Universal Robots PolyScope program: andrea8.urp

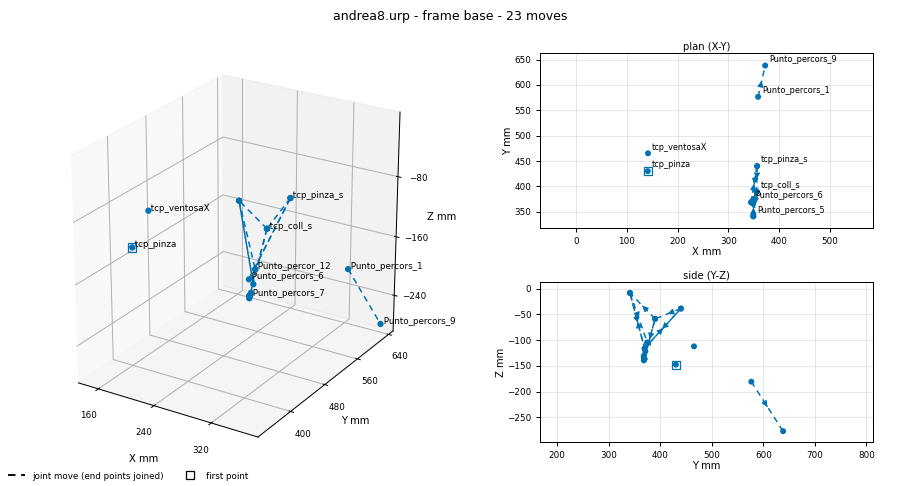
[picture p0: tool path of andrea8.urp in frame base, 23 of 31 moves have a stored position in this frame; points joined in program order, loops and branches not executed]
Program andrea8 (installation=Kong_install82 directory=/programs/usbdisk/andrea8 createdIn=3.15.4.106291 lastSavedIn=3.15.4.106291 robotSerialNumber=2017357596)
Calibrated DH parameters: a=[0.000104, -0.381245, -0.385946, 0.00002, 0.000083, 0]; d=[0.089177, 59.99214, -36.297918, -23.584132, 0.094784, 0.082552]; alpha=[1.570197, -0.003145, 0.002952, 1.570494, -1.570091, 0]; deltaTheta=[-0.00001, -0.459739, 0.638868, -0.17972, -0.000006, -0.000462]
InitVariablesNode variables(variable(name=XY, expression=[0,0]), variable(name=ant, expression=3), variable(name=col, expression=4), variable(name=ghr, expression=2), variable(name=nCycle, expression=0), variable(name=nfc, expression=1), variable(name=pallStocks, expression=[16,16,16,40,16,16,16,40,16,16,16,40,16,40,0,0]), variable(name=pick, expression=[0,0]))
Robot Program (runOnlyOnce=false)
  Script file /programs/usbdisk/andrea8/nuova dir/relPose.script
    | def relPose(FeaturePose,vect):
    | 
    |     # FeaturePose is the pose for the feature
    |     # vect = p[0.1, 0, 0, 0, 0, 0] makes us move 10cm in the X direction of the feature
    |     # credits: https://forum.universal-robots.com/t/move-tcp-relative-to-feature/15492
    | 
    |    PoseRelativeToFeature = pose_trans(pose_inv(FeaturePose), get_actual_tcp_pose())
    |    MoveTCPRelativeToFeature = pose_add(PoseRelativeToFeature, vect)
    |    return pose_trans(FeaturePose, MoveTCPRelativeToFeature)
    | 
    | end
  Script file /programs/usbdisk/andrea8/tcpMov.script
    | def tcpMov(vect):
    | 
    |     # FeaturePose is the pose for the feature
    |     # vect = p[0.1, 0, 0, 0, 0, 0] makes us move 10cm in the X direction of the feature
    |     # credits: https://forum.universal-robots.com/t/move-tcp-relative-to-feature/15492
    | 
    |    tcp_pose = get_actual_tcp_pose()
    |    return pose_add(tcp_pose, vect)
    | 
    | 
    | end
  Script file /programs/usbdisk/andrea8/calcItemPosition.script
    | def calcItemPosition(pick, item, pallDefs, grid, featOrigin):
    | 
    |     # calcola la posizione assoluta del pezzo scelto da pickPalletItem
    | 
    |     # nPosX è il numero di colonne
    |     # nPosY è il numero di righe
    |     # distX è la distanza tra colonne
    |     # distY è la distanza tra righe
    |     # [posX1, posY1] è la posizione del primo pezzo rispetto all'origine del pallet
    | 
    |     nPallet = pick[0] + 1 # numero del pallet (gli id partono da 0)
    |     nItem = pick[1] + 1 # numero del pezzo
    | 
    |     nPosXgrid = grid[0] # numero di posizioni della giglia in X
    |     distXgrid = grid[2] # distanza tra gli slot della griglia in X
    |     distYgrid = grid[3] # distanza tra gli slot della griglia in Y
    | 
    |     pallPosX = nPallet%nPosXgrid
    |     if(pallPosX==0): pallPosX = nPosXgrid end
    |     pallPosY = ceil(nPallet/nPosXgrid)
    | 
    |     pallPosX1 = grid[4]
    |     pallPosY1 = grid[5]
    | 
    | 
    |     nPosX = pallDefs[item,0]
    |     nPosY = pallDefs[item,1]
    |     distX = pallDefs[item,2]
    |     distY = pallDefs[item,3]
    |     posX1 = pallDefs[item,4]
    |     posY1 = pallDefs[item,5]
    | 
    |     posX = nItem%nPosX
    |     if(posX==0): posX = nPosX end
    |     posY = ceil(nItem/nPosX)
    | 
    |     # [X,Y] è la posizione del pezzo rispetto all'origine della griglia
    | 
    |     X=distX*(posX - 1) + posX1 + distXgrid*(pallPosX - 1) + pallPosX1
    |     Y=distY*(posY - 1) + posY1 + distYgrid*(pallPosY - 1) + pallPosY1
    |     xy=[X,Y]
    | 
    |     return xy
    | 
    |  end
  Script file /programs/usbdisk/andrea8/pickPalletItem.script
    | def pickPalletItem(type, pallDefs, pallTypes, pallStocks):
    | 
    |   # seleziona un pezzo sulla griglia, noti il tipo di pezzo e lo stato della griglia
    | 
    |   # lo script funziona finché le variabili del robot non vengono resettate. Tuttavia, anche
    |   # in caso di riavvio, è possibile scrivere manualmente le info sulla griglia e lo stock
    |   # all'inizio del programma, così da 'insegnare' al robot dove farlo
    |   # riprendere
    | 
    |   iPallet = 0 # inizializzo l'id del pallet
    | 
    |   while iPallet < length(pallStocks):
    | 
    |     if pallTypes[iPallet] == type and pallStocks[iPallet] > 0 :
    | 
    |       nItems = pallStocks[iPallet] # numero di pezzi nello stock del pallet iesimo
    | 
    |       nPosX = pallDefs[type,0] # numero di posizioni lungo x, come definito per il pallet di tipo "type"
    |       nPosY = pallDefs[type,1] # numero di posizioni lungo y, come definito per il pallet di tipo "type"
    | 
    |       stockMax = nPosX*nPosY
    |       iItem = stockMax - nItems # id del pezzo
    | 
    |       pick = [iPallet,iItem]
    | 
    |       # pick = [id del pallet, id del pezzo]
    | 
    |       return pick
    |  end
    | iPallet = iPallet + 1
    | end
    | end
  Script file /programs/usbdisk/andrea8/stockUpdate.script
    | def stockUpdate(pick,stock):
    | 
    |     # simple function that ingests the output of pickItem and returns the
    |     # modified stock array. just so to avoid using global variables and
    |     # multi-dimensional arrays
    | 
    |     i = pick[0]
    |     stock[i] = stock[i] - 1
    |     return stock
    | 
    | 
    | end
  SuppressedNode
    Script file /programs/usbdisk/andrea8/ini_grids.script
      | def ini_grids():
      | 
      |     # grid = [nPallPosX, nPallPosY, distPallX, distPallY, pallPosX1, pallPosY1, pallPosZ1]
      |     # la struttura e' del tutto analoga in logica con quella espressa in defs
      |     grids = [
      |                      [4, 4, 90, 90, 10, 20, 6] # griglia moduli
      |                      [2, 1, 200, 0, 20, -40, 45] # griglia stazioni
      |                  ]
      |     return grids
      | end
  Script file /programs/usbdisk/andrea8/ini_grid.script
    | def ini_grid():
    | 
    |     # grid = [nPallPosX, nPallPosY, distPallX, distPallY, pallPosX1, pallPosY1, pallPosZ1]
    |     # la struttura e' del tutto analoga in logica con quella espressa in defs
    |     grid = [4, 4, 90, 90, 10, 17.5, 6]
    |     return grid
    | end
  Script file /programs/usbdisk/andrea8/ini_defs.script
    | def ini_defs():
    | 
    |     # definition = [nPosX,nPosY,distX,distY,posX1,posY1,posZ1]
    | 
    |     # nPosX è il numero di colonne
    |     # nPosY è il numero di righe
    |     # distX è la distanza tra colonne
    |     # distY è la distanza tra righe
    |     # [posX1, posY1] è la posizione del primo pezzo rispetto all'origine del pallet
    |     # posZ1 e' la posizione che deve raggiungere il TCP lungo asse Z, che sarebbe asse verticale
    | 
    |     defs = [
    |         [0, 0, 0, 0, 0, 0, 0], # slot vuoto
    |         [4, 10, 18, 8, 11.5, 3.5, 11.1], # pallet nfc
    |         [4, 4, 21, 21, 5.5, 8.5, 49], # pallet ghiere
    |         [1, 1, 0, 0, 132.06, 44, 16.05], # stazione antenna
    |         [1, 2, 0, 40, 20.256, 24, 27.85] # stazione incollaggio
    |     ]
    |     return defs
    | end
  Script file /programs/usbdisk/andrea8/ini_types.script
    | def ini_types():
    | 
    |     visualTypes = [
    | 
    |         [0,0,0,0],
    |         [0,ghr,0,0],
    |         [0,0,0,nfc],
    |         [0,ghr,0,0]
    | 
    |     ]
    | 
    | # purtroppo fare questa array vuota di dimensione (righe)x(colonne) per aggirare le limitazioni di UR
    | # bisogna ricordarsi di cambiare questa dichiarazione di types se si cambia dimensione griglia
    | 
    |      types = [0,0,0,0,0,0,0,0,0,0,0,0,0,0,0,0]
    | 
    |     iii = 0
    |     s = size(visualTypes)
    |     i = 0
    |     while i < s[0]:
    | 
    |         ii=0
    |         while ii < s[1]:
    | 
    |             types[iii] = visualTypes[s[0]-1-i,ii]
    |             ii = ii + 1
    |             iii = iii + 1
    |         end
    |     i = i + 1
    |     end
    |     return types
    | end
  Script file /programs/usbdisk/andrea8/ini_stocks2.script
    | def ini_stocks(defs, types):
    | 
    |     global f = -1 # usa questo carattere per inizializzare automaticamente pallet pieni
    | 
    |     visualStocks = [
    | 
    |         [f, f, f, f],
    |         [f, f, f, f],
    |         [f, f, f, 36],
    |         [f ,f, f, f]
    | 
    |     ]
    | 
    | # purtroppo fare questa array vuota di dimensione (righe)x(colonne) per aggirare le limitazioni di UR
    | # bisogna ricordarsi di cambiare questa dichiarazione di types se si cambia dimensione griglia
    | 
    |      stocks = [0,0,0,0,0,0,0,0,0,0,0,0,0,0,0,0]
    | 
    |     iii = 0
    |     s = size(visualStocks)
    |     i = 0
    |     while i < s[0]:
    | 
    |         ii=0
    |         while ii < s[1]:
    |             if visualStocks[s[0]-1-i,ii] == f:
    |                 nPosX = defs[types[iii], 0]
    |                 nPosY = defs[types[iii], 1]
    |                 stocks[iii] = nPosX*nPosY
    |             else:
    | 
    |                 stocks[iii] = visualStocks[s[0]-1-i,ii]
    |             end
    |             ii = ii + 1
    |             iii = iii + 1
    |         end
    |     i = i + 1
    |     end
    |     return stocks
    | end
  If nCycle≟0
    Set NoAction
    pallTypes := ini_types()
    grid := ini_grid()
    pallDefs := ini_defs()
    pallStocks := ini_stocks(pallDefs,pallTypes)
    SuppressedNode
      Popup Message (haltProgram=false inputType=Variable) variable=grid
    ghr := ghr
    nfc := nfc
    ant := ant
    col := col
    URCap Open Gripper (SCHUNK End-of-Arm Modular System for UR, SCHUNK GmbH & Co.)
    nCycle := 1
    Wait Sleep waitTime=5
  MoveJ speed 60 deg/s, acceleration 80 deg/s^2 (useActiveTCP=false) tcp=Pinza
    Waypoint tcp_pinza: TCP in base x=141.498 y=430.173 z=-147.715 mm, rx=-2.3787 ry=0.7214 rz=1.7108 rad; joints [-125.948, -50.519, 103.828, -113.29, -23.958, -21.608] deg; pose in feature x=-0.012 y=-0.048 z=150.016 mm, rx=-1.1212 ry=1.1212 rz=0.4102 rad; flange x=182.463 y=570.54 z=26.56 mm, rx=-2.3787 ry=0.7214 rz=1.7108 rad
    item := ghr
    pick := pickPalletItem(item,pallDefs,pallTypes,pallStocks)
    SuppressedNode
      Popup Message (haltProgram=false inputType=Variable) variable=pick
    XY := calcItemPosition(pick, item,pallDefs, grid,piano_moduli)
    p_pall := relPose(piano_moduli,p[XY[0]/1000,XY[1]/1000,0.0,0.0,0.0,0.0])
    SuppressedNode
      Popup Message (haltProgram=false inputType=Variable) variable=XY
    Waypoint Punto_percors (Variable): variable=p_pall
  MoveJ speed 60 deg/s, acceleration 80 deg/s^2 (useActiveTCP=false) tcp=Pinza
    p_pezzo := relPose(piano_moduli,p[0.0, 0.0, -130*0.001, 0.0, 0.0, 0.0])
    Waypoint Punto_percors (Variable): variable=p_pezzo
    URCap Close Gripper (SCHUNK End-of-Arm Modular System for UR, SCHUNK GmbH & Co.)
    p_pezzo := relPose(piano_moduli,p[0.0, 0.0, 130/1000, 0.0, 0.0, 0.0])
    Waypoint Punto_percors (Variable): variable=p_pezzo
    pallStocks := stockUpdate(pick,pallStocks)
    SuppressedNode
      Popup Message (haltProgram=false inputType=Variable) variable=pallStocks
  MoveJ speed 60 deg/s, acceleration 80 deg/s^2 (useActiveTCP=false) tcp=Ventosa
    Waypoint tcp_ventosaX: TCP in base x=141.953 y=465.356 z=-112.213 mm, rx=-2.2886 ry=-0.6046 rz=-0.263 rad; joints [-121.609, -49.485, 100.63, -2.12, 68.781, 127.146] deg; flange x=141.931 y=500.256 z=-13.059 mm, rx=-2.2886 ry=-0.6046 rz=-0.263 rad
    SuppressedNode
      Waypoint tcp_ventosaY_s: TCP in base x=355.984 y=389.916 z=-58.857 mm, rx=-1.401 ry=-1.0647 rz=1.3858 rad; joints [-146.472, -36.177, 73.345, -37.097, -55.375, 194.745] deg; pose in feature x=141.985 y=465.345 z=-112.215 mm, rx=-1.4011 ry=-1.0646 rz=1.3857 rad; flange x=401.93 y=456.119 z=8.64 mm, rx=-1.401 ry=-1.0647 rz=1.3858 rad
    item := nfc
    pick := pickPalletItem(item,pallDefs,pallTypes,pallStocks)
    SuppressedNode
      Popup Message (haltProgram=false inputType=Variable) variable=pick
    XY := calcItemPosition(pick, item,pallDefs, grid,piano_moduli)
    p_pall := relPose(piano_moduli,p[XY[0]/1000,XY[1]/1000,0.0,0.0,0.0,0.0])
    SuppressedNode
      Popup Message (haltProgram=false inputType=Variable) variable=XY
    Waypoint Punto_percors (Variable): variable=p_pall
  MoveJ speed 60 deg/s, acceleration 80 deg/s^2 (useActiveTCP=false) tcp=Ventosa
    p_pezzo := relPose(piano_moduli,p[0.0, 0.0, -181.4*0.001, 0.0, 0.0, 0.0])
    Waypoint Punto_percors (Variable): variable=p_pezzo
    Wait Sleep waitTime=2
    p_pezzo := relPose(piano_moduli,p[0.0, 0.0, 181.4/1000, 0.0, 0.0, 0.0])
    Waypoint Punto_percors (Variable): variable=p_pezzo
    pallStocks := stockUpdate(pick,pallStocks)
    SuppressedNode
      Popup Message (haltProgram=false inputType=Variable) variable=pallStocks
  MoveJ speed 60 deg/s, acceleration 80 deg/s^2 (useActiveTCP=false) tcp=Ventosa
    Waypoint Punto_percors_1: TCP in base x=358.691 y=576.543 z=-180.701 mm, rx=-2.2887 ry=-0.6045 rz=-0.2628 rad; joints [-132.678, -21.575, 54.335, 20.288, 61.783, 117.598] deg; flange x=358.684 y=611.454 z=-81.55 mm, rx=-2.2887 ry=-0.6045 rz=-0.2628 rad
    Waypoint Punto_percors_9: TCP in base x=372.703 y=638.173 z=-276.765 mm, rx=-2.2781 ry=-0.6995 rz=-0.1741 rad; joints [-130.314, 4.573, 13.616, 38.475, 59.716, 114.972] deg; flange x=372.486 y=675.646 z=-178.554 mm, rx=-2.2781 ry=-0.6995 rz=-0.1741 rad
    SuppressedNode
      MoveJ speed 60 deg/s, acceleration 80 deg/s^2 (useActiveTCP=true)
        Waypoint Punto_percors_2: 
  MoveJ speed 60 deg/s, acceleration 80 deg/s^2 (useActiveTCP=false) tcp=Ventosa
    p_pezzo := relPose(piano_moduli,p[0.0, 0.0, -55*0.001, 0.0, 0.0, 0.0])
    Waypoint Punto_percors (Variable): variable=p_pezzo
    Wait Sleep waitTime=2
    p_pezzo := relPose(piano_moduli,p[0.0, 0.0, 55/1000, 0.0, 0.0, 0.0])
    Waypoint Punto_percors (Variable): variable=p_pezzo
  MoveJ speed 60 deg/s, acceleration 80 deg/s^2 (useActiveTCP=false) tcp=Pinza
    Waypoint tcp_pinza_s: TCP in base x=356.783 y=439.979 z=-38.857 mm, rx=1.9379 ry=-1.1643 rz=-1.0823 rad; joints [-132.207, -20.407, 45.734, -60.67, -53.979, 1] deg; flange x=387.119 y=665.322 z=-46.123 mm, rx=1.9379 ry=-1.1643 rz=-1.0823 rad
    Waypoint Punto_percors_6: TCP in base x=344.955 y=369.152 z=-116.441 mm, rx=1.9235 ry=-1.2186 rz=-1.1045 rad; joints [-136.086, -22.163, 63.024, -76.094, -54.959, 0.389] deg; flange x=386.118 y=592.787 z=-123.208 mm, rx=1.9235 ry=-1.2186 rz=-1.1045 rad
    URCap Open Gripper (SCHUNK End-of-Arm Modular System for UR, SCHUNK GmbH & Co.)
    Waypoint tcp_pinza_s: TCP in base x=356.783 y=439.979 z=-38.857 mm, rx=1.9379 ry=-1.1643 rz=-1.0823 rad; joints [-132.207, -20.407, 45.734, -60.67, -53.979, 1] deg; flange x=387.119 y=665.322 z=-46.123 mm, rx=1.9379 ry=-1.1643 rz=-1.0823 rad
  SuppressedNode
    MoveJ speed 60 deg/s, acceleration 80 deg/s^2 (useActiveTCP=false) tcp=Pinza
      p_pezzo := relPose(piano_moduli,p[0.0, 0.0, -100*0.001, 0.0, 0.0, 0.0])
      Waypoint Punto_percors (Variable): variable=p_pezzo
      p_pezzo := relPose(piano_moduli,p[0.0, 0.0, 100/1000, 0.0, 0.0, 0.0])
      Waypoint Punto_percors (Variable): variable=p_pezzo
  MoveJ speed 60 deg/s, acceleration 80 deg/s^2 (useActiveTCP=false) tcp=Dosatore_Colla
    Waypoint tcp_coll_s: TCP in base x=355.98 y=389.944 z=-58.821 mm, rx=-0.0221 ry=-3.1138 rz=0.4025 rad; joints [-139.161, -64.308, 106.34, -121.985, -100.827, 102.96] deg; flange x=356.624 y=435.245 z=113.503 mm, rx=0.7684 ry=-2.9515 rz=0.3801 rad
    Waypoint Punto_percors_7: TCP in base x=346.196 y=368.904 z=-136.542 mm, rx=-0.022 ry=-3.1138 rz=0.4025 rad; joints [-139.88, -59.505, 111.836, -132.417, -100.987, 102.258] deg; flange x=346.894 y=417.717 z=49.148 mm, rx=0.7685 ry=-2.9514 rz=0.38 rad
    Waypoint Punto_percors_8: TCP in base x=346.193 y=368.067 z=-139.507 mm, rx=-0.0222 ry=-3.1137 rz=0.4027 rad; joints [-139.945, -59.217, 112.004, -132.878, -101.004, 102.201] deg; flange x=346.901 y=416.902 z=46.177 mm, rx=0.7683 ry=-2.9514 rz=0.3802 rad
    Waypoint Punto_percors_7: TCP in base x=346.196 y=368.904 z=-136.542 mm, rx=-0.022 ry=-3.1138 rz=0.4025 rad; joints [-139.88, -59.505, 111.836, -132.417, -100.987, 102.258] deg; flange x=346.894 y=417.717 z=49.148 mm, rx=0.7685 ry=-2.9514 rz=0.38 rad
    Waypoint arco01: TCP in base x=346.236 y=368.89 z=-136.518 mm, rx=-0.0959 ry=-3.05 rz=0.3936 rad; joints [-141.187, -58.835, 109.658, -128.209, -98.558, 103.729] deg; flange x=360.097 y=417.145 z=48.801 mm, rx=0.6834 ry=-2.9135 rz=0.3475 rad
    Waypoint arco02: motionParameters(blendRadius=0); TCP in base x=346.216 y=368.872 z=-136.545 mm, rx=-0.179 ry=-2.9723 rz=0.3829 rad; joints [-142.748, -57.872, 107.148, -123.504, -95.68, 105.297] deg; flange x=375.525 y=415.536 z=47.377 mm, rx=0.5857 ry=-2.8653 rz=0.31 rad
    Waypoint arco03: motionParameters(blendRadius=0); TCP in base x=346.203 y=368.894 z=-136.515 mm, rx=-0.2657 ry=-2.8849 rz=0.3708 rad; joints [-144.474, -56.651, 104.495, -118.647, -92.526, 106.837] deg; flange x=392.12 y=412.637 z=44.709 mm, rx=0.482 ry=-2.8087 rz=0.2699 rad
    SuppressedNode
      Waypoint arco04: motionParameters(blendRadius=0); TCP in base x=346.203 y=368.881 z=-136.572 mm, rx=-0.3164 ry=-2.8302 rz=0.3633 rad; joints [-145.538, -55.821, 102.932, -115.817, -90.6, 107.69] deg; flange x=402.069 y=410.254 z=42.401 mm, rx=0.4203 ry=-2.7721 rz=0.2459 rad
    SuppressedNode
      Waypoint arrco05: motionParameters(blendRadius=0); TCP in base x=346.234 y=368.906 z=-136.515 mm, rx=-0.3852 ry=-2.7521 rz=0.3526 rad; joints [-147.033, -54.592, 100.815, -111.993, -87.907, 108.809] deg; flange x=415.666 y=406.217 z=38.559 mm, rx=0.3354 ry=-2.7188 rz=0.2129 rad
    SuppressedNode
      Waypoint arco06: motionParameters(blendRadius=0); TCP in base x=346.215 y=368.872 z=-136.573 mm, rx=-0.447 ry=-2.677 rz=0.3424 rad; joints [-148.443, -53.359, 98.932, -108.559, -85.383, 109.759] deg; flange x=427.962 y=401.606 z=34.043 mm, rx=0.2577 ry=-2.666 rz=0.1826 rad
    SuppressedNode
      Waypoint arco07: motionParameters(blendRadius=0); TCP in base x=346.221 y=368.89 z=-136.541 mm, rx=-0.508 ry=-2.5984 rz=0.3316 rad; joints [-149.891, -52.049, 97.106, -105.173, -82.796, 110.659] deg; flange x=440.036 y=396.148 z=28.747 mm, rx=0.1797 ry=-2.6097 rz=0.1519 rad
    SuppressedNode
      Waypoint arco08: motionParameters(blendRadius=0); TCP in base x=346.175 y=368.881 z=-136.554 mm, rx=-0.5601 ry=-2.5271 rz=0.322 rad; joints [-151.177, -50.841, 95.583, -102.267, -80.5, 111.395] deg; flange x=450.208 y=390.667 z=23.341 mm, rx=0.1118 ry=-2.5574 rz=0.1253 rad
    SuppressedNode
      Waypoint arco07: motionParameters(blendRadius=0); TCP in base x=346.221 y=368.89 z=-136.541 mm, rx=-0.508 ry=-2.5984 rz=0.3316 rad; joints [-149.891, -52.049, 97.106, -105.173, -82.796, 110.659] deg; flange x=440.036 y=396.148 z=28.747 mm, rx=0.1797 ry=-2.6097 rz=0.1519 rad
    SuppressedNode
      Waypoint arco06: motionParameters(blendRadius=0); TCP in base x=346.215 y=368.872 z=-136.573 mm, rx=-0.447 ry=-2.677 rz=0.3424 rad; joints [-148.443, -53.359, 98.932, -108.559, -85.383, 109.759] deg; flange x=427.962 y=401.606 z=34.043 mm, rx=0.2577 ry=-2.666 rz=0.1826 rad
    SuppressedNode
      Waypoint arrco05: motionParameters(blendRadius=0); TCP in base x=346.234 y=368.906 z=-136.515 mm, rx=-0.3852 ry=-2.7521 rz=0.3526 rad; joints [-147.033, -54.592, 100.815, -111.993, -87.907, 108.809] deg; flange x=415.666 y=406.217 z=38.559 mm, rx=0.3354 ry=-2.7188 rz=0.2129 rad
    SuppressedNode
      Waypoint arco04: motionParameters(blendRadius=0); TCP in base x=346.203 y=368.881 z=-136.572 mm, rx=-0.3164 ry=-2.8302 rz=0.3633 rad; joints [-145.538, -55.821, 102.932, -115.817, -90.6, 107.69] deg; flange x=402.069 y=410.254 z=42.401 mm, rx=0.4203 ry=-2.7721 rz=0.2459 rad
    SuppressedNode
      Waypoint arco03: motionParameters(blendRadius=0); TCP in base x=346.203 y=368.894 z=-136.515 mm, rx=-0.2657 ry=-2.8849 rz=0.3708 rad; joints [-144.474, -56.651, 104.495, -118.647, -92.526, 106.837] deg; flange x=392.12 y=412.637 z=44.709 mm, rx=0.482 ry=-2.8087 rz=0.2699 rad
    Waypoint arco02: motionParameters(blendRadius=0); TCP in base x=346.216 y=368.872 z=-136.545 mm, rx=-0.179 ry=-2.9723 rz=0.3829 rad; joints [-142.748, -57.872, 107.148, -123.504, -95.68, 105.297] deg; flange x=375.525 y=415.536 z=47.377 mm, rx=0.5857 ry=-2.8653 rz=0.31 rad
    Waypoint arco01: TCP in base x=346.236 y=368.89 z=-136.518 mm, rx=-0.0959 ry=-3.05 rz=0.3936 rad; joints [-141.187, -58.835, 109.658, -128.209, -98.558, 103.729] deg; flange x=360.097 y=417.145 z=48.801 mm, rx=0.6834 ry=-2.9135 rz=0.3475 rad
    Waypoint tcp_coll_s: TCP in base x=355.98 y=389.944 z=-58.821 mm, rx=-0.0221 ry=-3.1138 rz=0.4025 rad; joints [-139.161, -64.308, 106.34, -121.985, -100.827, 102.96] deg; flange x=356.624 y=435.245 z=113.503 mm, rx=0.7684 ry=-2.9515 rz=0.3801 rad
    SuppressedNode
      Waypoint tcp_colla: TCP in base x=141.953 y=465.356 z=-112.213 mm, rx=-0.0207 ry=-2.9002 rz=1.1933 rad; joints [-112.251, -46.475, 88.048, -88.757, -104.681, 134.691] deg; flange x=143.75 y=590.738 z=14.373 mm, rx=0.6882 ry=-2.6438 rz=1.0836 rad
  MoveJ speed 60 deg/s, acceleration 80 deg/s^2 (useActiveTCP=false) tcp=Ventosa
    Waypoint Punto_percors_5: TCP in base x=349.319 y=341.12 z=-8.564 mm, rx=-1.0185 ry=-1.3146 rz=1.0001 rad; joints [-153.414, -49.535, 86.3, -36.662, -62.309, 164.702] deg; flange x=394.672 y=364.631 z=83.305 mm, rx=-1.0185 ry=-1.3146 rz=1.0001 rad
    Waypoint Punto_percor_11: TCP in base x=349.675 y=371.112 z=-122.13 mm, rx=-1.0185 ry=-1.3145 rz=1.0002 rad; joints [-150.91, -37.388, 83.592, -46.127, -59.801, 164.771] deg; flange x=395.037 y=394.636 z=-30.269 mm, rx=-1.0185 ry=-1.3145 rz=1.0002 rad
    Wait Sleep waitTime=1
    Waypoint Punto_percors_5: TCP in base x=349.319 y=341.12 z=-8.564 mm, rx=-1.0185 ry=-1.3146 rz=1.0001 rad; joints [-153.414, -49.535, 86.3, -36.662, -62.309, 164.702] deg; flange x=394.672 y=364.631 z=83.305 mm, rx=-1.0185 ry=-1.3146 rz=1.0001 rad
    SuppressedNode
      Waypoint tcp_ventosaY_s: TCP in base x=355.984 y=389.916 z=-58.857 mm, rx=-1.401 ry=-1.0647 rz=1.3858 rad; joints [-146.472, -36.177, 73.345, -37.097, -55.375, 194.745] deg; flange x=401.93 y=456.119 z=8.64 mm, rx=-1.401 ry=-1.0647 rz=1.3858 rad
    SuppressedNode
      Waypoint Punto_percors_4: 
  MoveJ speed 60 deg/s, acceleration 80 deg/s^2 (useActiveTCP=false) tcp=Pressa
    Waypoint Punto_percor_12: TCP in base x=349.834 y=374.867 z=-104.947 mm, rx=0.1982 ry=-1.5625 rz=-0.2204 rad; joints [-149.184, -43.549, 79.977, -36.342, -58.078, 74.726] deg; flange x=395.431 y=416.173 z=54.625 mm, rx=0.1982 ry=-1.5625 rz=-0.2204 rad
    Waypoint Punto_percor_13: TCP in base x=348.512 y=367.85 z=-131.982 mm, rx=0.1982 ry=-1.5627 rz=-0.2205 rad; joints [-149.684, -41.891, 81.658, -39.702, -58.567, 74.74] deg; flange x=394.082 y=409.131 z=27.605 mm, rx=0.1982 ry=-1.5627 rz=-0.2205 rad
    Wait Sleep waitTime=2
    Waypoint Punto_percor_12: TCP in base x=349.834 y=374.867 z=-104.947 mm, rx=0.1982 ry=-1.5625 rz=-0.2204 rad; joints [-149.184, -43.549, 79.977, -36.342, -58.078, 74.726] deg; flange x=395.431 y=416.173 z=54.625 mm, rx=0.1982 ry=-1.5625 rz=-0.2204 rad
    SuppressedNode
      Waypoint tcp_pressaY: TCP in base x=141.469 y=430.16 z=-147.709 mm, rx=-0.2128 ry=-1.5595 rz=0.1907 rad; joints [-127.014, -38.383, 85.876, -47.443, -35.896, 104.766] deg; flange x=188.109 y=545.63 z=-30.49 mm, rx=-0.2128 ry=-1.5595 rz=0.1907 rad
    SuppressedNode
      Waypoint tcp_pressaX: TCP in base x=141.415 y=430.194 z=-147.729 mm, rx=-1.3127 ry=-2.237 rz=-0.9404 rad; joints [-120.759, -49.8, 97.992, 0.536, 69.418, 38.219] deg; flange x=142.623 y=514.321 z=1.167 mm, rx=-1.3127 ry=-2.237 rz=-0.9404 rad
  SuppressedNode
    Popup Message (haltProgram=false inputType=Variable) variable=pick
